{attribute 'linkalways'} 
{attribute 'no_explicit_call' := 'This FB is a CLASS and must be accessed using methods or properties'}
{attribute 'enable_dynamic_creation'}
FUNCTION_BLOCK FINAL ACOS_LREAL EXTENDS Node
VAR
	in : _LREAL(0.0);
	out : _LREAL(0.0);
END_VAR

METHOD PUBLIC Clone : I_Node
VAR
	pNode : POINTER TO ACOS_LREAL;
END_VAR
pNode := __NEW(ACOS_LREAL);
Clone := pNode^;
END_METHOD

METHOD FB_init : BOOL
VAR_INPUT
	bInitRetains : BOOL; // if TRUE, the retain variables are initialized (warm start / cold start)
	bInCopyCode : BOOL;  // if TRUE, the instance afterwards gets moved into the copy code (online change)
END_VAR
AddInput('in',THIS^.in);
AddOutput('out', THIS^.out);
END_METHOD

METHOD PROTECTED OnExecute
VAR
END_VAR
out.Value := ACOS(in.Value);
END_METHOD

END_FUNCTION_BLOCK

(* stored: Version 1.1.0.1, ProductVersion 3.1.4024.15
   POU ACOS_LREAL: Id {0ba0ece8-f80e-4b6b-a64f-418922df5262}, SpecialFunc None
   Folder Constructor: Id {1f0f9f1b-4199-4406-bfd5-eeed1edf6497}
   Method Clone: Id {8c58fc39-d556-4f28-9ab1-e3d155419dcd}
   Method FB_init: Id {bd06a6f2-fb75-4bea-8b1e-60020d05e625}
   Method OnExecute: Id {aae94cec-f32e-42a0-acce-0319043bd3b4} *)
